Staubli VAL3: COGNEX2.pjx

Parameters version=s7.6 stackSize=5000 millimeterUnit=true
Program file=create.pgx
Program file=detection.pgx
Program file=getMaxNumOfPart.pgx
Program file=getObjectData.pgx
Program file=getObjectLatch.pgx
Program file=init.pgx
Program file=initvis.pgx
Program file=isDetected.pgx
Program file=kill.pgx
Program file=resetTask.pgx
Program file=sortObjects.pgx
Program file=start.pgx
Program file=stop.pgx
Data file=Cognex2.dtx
Library alias=ut path=Disk://Tracking/Tools/util/util.pjx
Library alias=cam path=./cognexComm/cognexComm.pjx
Library alias=sck path=Disk://Tracking/io/sockets/sockets.pjx
Type name=object path=Disk://Tracking/Templates/object/object.pjx
